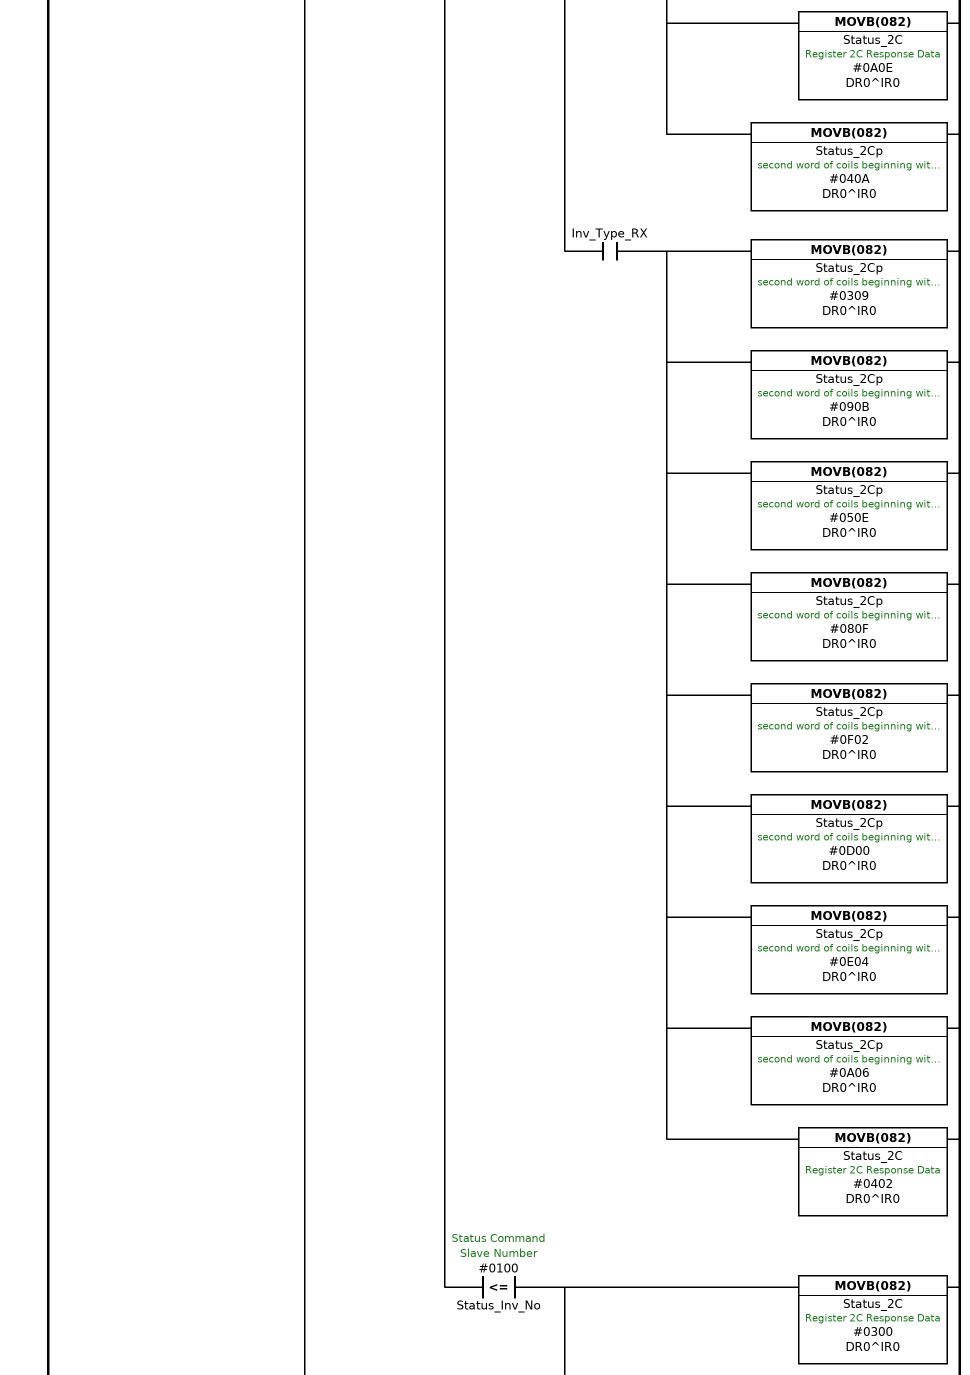
; [picture p48: FB INV002_Refresh_X31_, rungs 31-31]

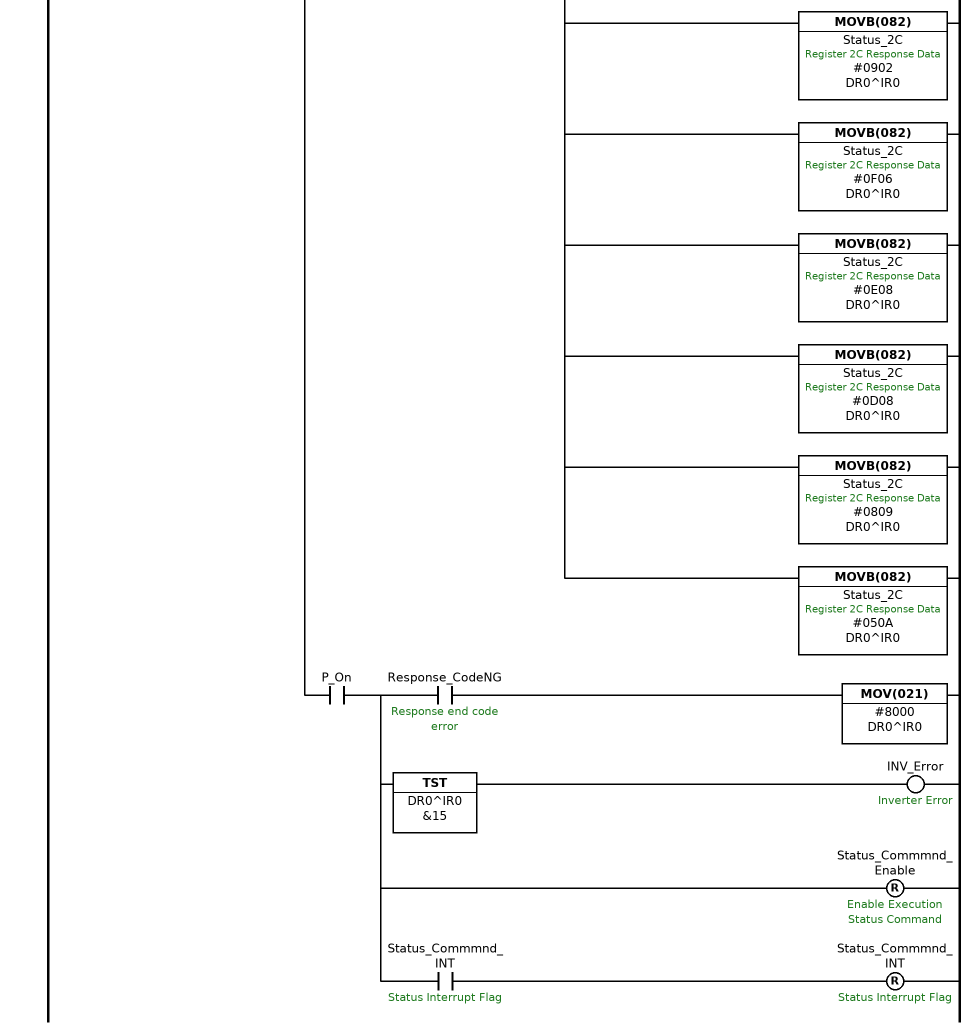
; rung 31: Generate Status Process
LD Status_Commmnd_Enable  ; Enable Execution Status Command
AND=(300) &3 Phase  ; Process Procedure
OUT TR0
AND P_On
MOV(021) Status_Inv_No Tmp_Data[0]  ; Status Command Slave Number
ANDW(034) Tmp_Data[0] #00FF Tmp_Data[0]
-(410) Tmp_Data[0] &1 Tmp_Data[0]
*(420) Tmp_Data[0] &2 Tmp_Data[0]
MOV(021) Tmp_Data[0] DR0
LD TR0
ANDNOT Response_CodeNG  ; Response end code error
OUT TR1
AND>(320) #0100 Status_Inv_No  ; Status Command Slave Number
OUT TR2
ANDNOT Inv_Type_RX
MOVB(082) Status_2C #0301 DR0^IR0  ; Register 2C Response Data
MOVB(082) Status_2C #0903 DR0^IR0  ; Register 2C Response Data
MOVB(082) Status_2C #0506 DR0^IR0  ; Register 2C Response Data
MOVB(082) Status_2C #0807 DR0^IR0  ; Register 2C Response Data
MOVB(082) Status_2C #0F0A DR0^IR0  ; Register 2C Response Data
MOVB(082) Status_2C #0D08 DR0^IR0  ; Register 2C Response Data
MOVB(082) Status_2C #0E0C DR0^IR0  ; Register 2C Response Data
MOVB(082) Status_2C #0A0E DR0^IR0  ; Register 2C Response Data
MOVB(082) Status_2Cp #040A DR0^IR0  ; second word of coils beginning with coil 1F to 2E
LD TR2
AND Inv_Type_RX
MOVB(082) Status_2Cp #0309 DR0^IR0  ; second word of coils beginning with coil 1F to 2E
MOVB(082) Status_2Cp #090B DR0^IR0  ; second word of coils beginning with coil 1F to 2E
MOVB(082) Status_2Cp #050E DR0^IR0  ; second word of coils beginning with coil 1F to 2E
MOVB(082) Status_2Cp #080F DR0^IR0  ; second word of coils beginning with coil 1F to 2E
MOVB(082) Status_2Cp #0F02 DR0^IR0  ; second word of coils beginning with coil 1F to 2E
MOVB(082) Status_2Cp #0D00 DR0^IR0  ; second word of coils beginning with coil 1F to 2E
MOVB(082) Status_2Cp #0E04 DR0^IR0  ; second word of coils beginning with coil 1F to 2E
MOVB(082) Status_2Cp #0A06 DR0^IR0  ; second word of coils beginning with coil 1F to 2E
MOVB(082) Status_2C #0402 DR0^IR0  ; Register 2C Response Data
LD TR1
AND<=(315) #0100 Status_Inv_No  ; Status Command Slave Number
MOVB(082) Status_2C #0300 DR0^IR0  ; Register 2C Response Data
MOVB(082) Status_2C #0902 DR0^IR0  ; Register 2C Response Data
MOVB(082) Status_2C #0F06 DR0^IR0  ; Register 2C Response Data
MOVB(082) Status_2C #0E08 DR0^IR0  ; Register 2C Response Data
MOVB(082) Status_2C #0D08 DR0^IR0  ; Register 2C Response Data
MOVB(082) Status_2C #0809 DR0^IR0  ; Register 2C Response Data
MOVB(082) Status_2C #050A DR0^IR0  ; Register 2C Response Data
LD TR0
AND P_On
OUT TR3
AND Response_CodeNG  ; Response end code error
MOV(021) #8000 DR0^IR0
LD TR3
ANDTST(350) DR0^IR0 &15
OUT INV_Error  ; Inverter Error
LD TR3
RSET Status_Commmnd_Enable  ; Enable Execution Status Command
AND Status_Commmnd_INT  ; Status Interrupt Flag
RSET Status_Commmnd_INT  ; Status Interrupt Flag

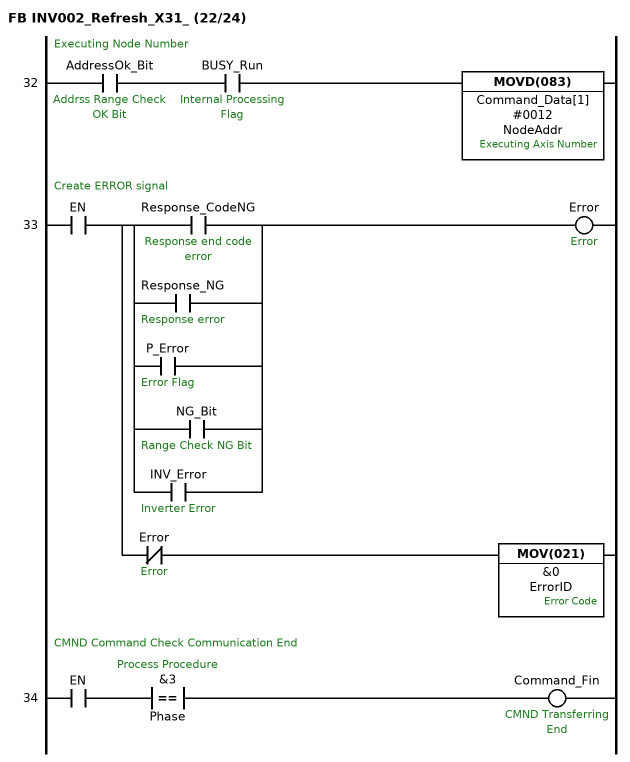
; rung 32: Executing Node Number
LD AddressOk_Bit  ; Addrss Range Check OK Bit
AND BUSY_Run  ; Internal Processing Flag
MOVD(083) Command_Data[1] #0012 NodeAddr  ; Executing Axis Number
; rung 33: Create ERROR signal
LD EN
OUT TR0
LD Response_CodeNG  ; Response end code error
OR Response_NG  ; Response error
OR P_Error  ; Error Flag
OR NG_Bit  ; Range Check NG Bit
OR INV_Error  ; Inverter Error
ANDLD
OUT Error  ; Error
LD TR0
ANDNOT Error  ; Error
MOV(021) &0 ErrorID  ; Error Code
; rung 34: CMND Command Check Communication End
LD EN
AND=(300) &3 Phase  ; Process Procedure
OUT Command_Fin  ; CMND Transferring End

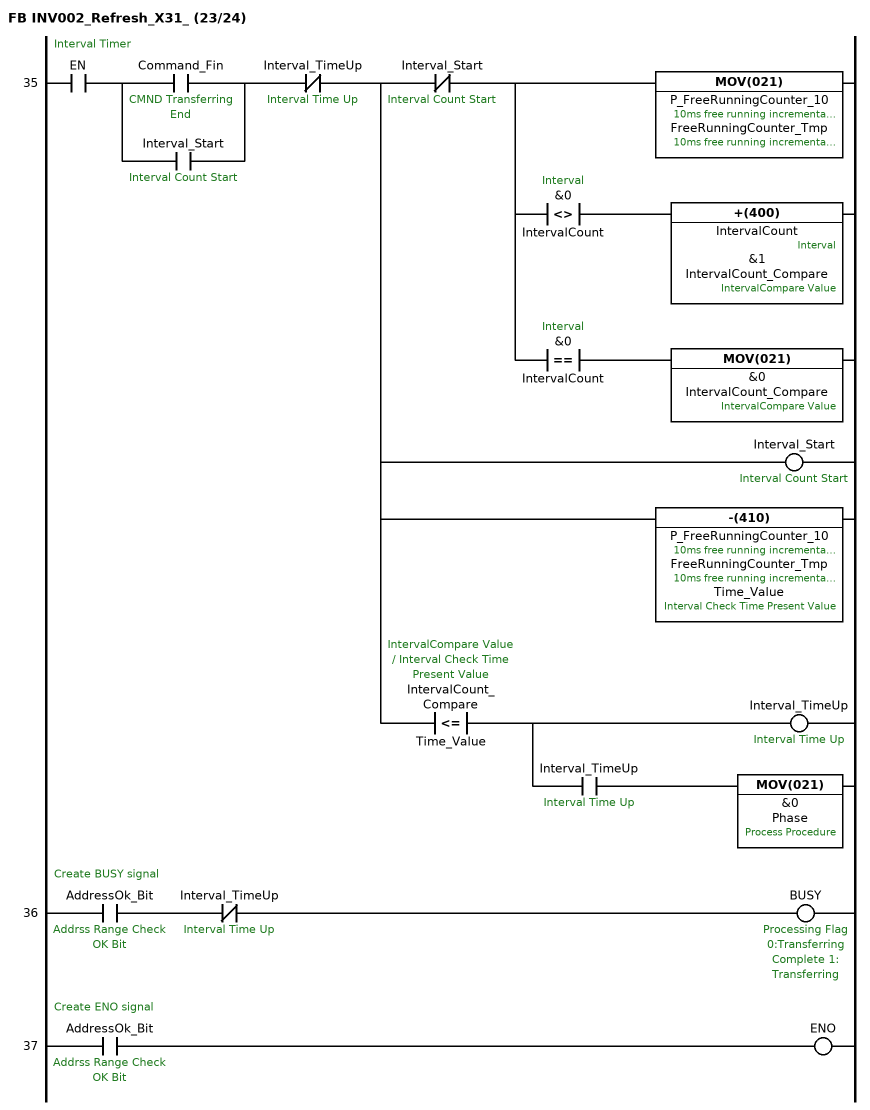
; rung 35: Interval Timer
LD EN
LD Command_Fin  ; CMND Transferring End
OR Interval_Start  ; Interval Count Start
ANDLD
ANDNOT Interval_TimeUp  ; Interval Time Up
OUT TR0
ANDNOT Interval_Start  ; Interval Count Start
OUT TR1
MOV(021) P_FreeRunningCounter_10 FreeRunningCounter_Tmp  ; 10ms free running incremental counter, 10ms free running incremental counter record
AND<>(305) &0 IntervalCount  ; Interval
+(400) IntervalCount &1 IntervalCount_Compare  ; Interval, IntervalCompare Value
LD TR1
AND=(300) &0 IntervalCount  ; Interval
MOV(021) &0 IntervalCount_Compare  ; IntervalCompare Value
LD TR0
OUT Interval_Start  ; Interval Count Start
-(410) P_FreeRunningCounter_10 FreeRunningCounter_Tmp Time_Value  ; 10ms free running incremental counter, 10ms free running incremental counter record, Interval Check Time Present Value
AND<=(315) IntervalCount_Compare Time_Value  ; IntervalCompare Value, Interval Check Time Present Value
OUT Interval_TimeUp  ; Interval Time Up
AND Interval_TimeUp  ; Interval Time Up
MOV(021) &0 Phase  ; Process Procedure
; rung 36: Create BUSY signal
LD AddressOk_Bit  ; Addrss Range Check OK Bit
ANDNOT Interval_TimeUp  ; Interval Time Up
OUT BUSY  ; Processing Flag 0:Transferring Complete 1:Transferring
; rung 37: Create ENO signal
LD AddressOk_Bit  ; Addrss Range Check OK Bit
OUT ENO

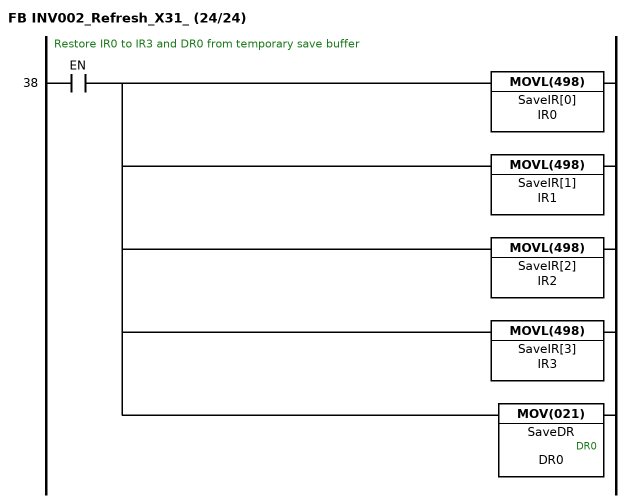
; rung 38: Restore IR0 to IR3 and DR0 from temporary save buffer
LD EN
MOVL(498) SaveIR[0] IR0
MOVL(498) SaveIR[1] IR1
MOVL(498) SaveIR[2] IR2
MOVL(498) SaveIR[3] IR3
MOV(021) SaveDR DR0  ; DR0

## Function block Новый_день
VAR_INPUT
  Day_star : UINT;
  Day_onl : UINT;
  Mon_star : UINT;
  Mon_onl : UINT;
  Day2 : UINT;
  Day3 : UINT;
  Mon2 : UINT;
  Mon3 : UINT;
END_VAR
VAR_OUTPUT
  Day_new : UINT;
  Mon_new : UINT;
  DayOut1 : UINT;
  DayOut2 : UINT;
  DayOut3 : UINT;
  MonOut1 : UINT;
  MonOut2 : UINT;
  MonOut3 : UINT;
END_VAR
	DayOut1 := Day2; DayOut2 := Day3; DayOut3 := Day_star;
	MonOut1 := Mon2; MonOut2 := Mon3; MonOut3 := Mon_star;
	Mon_new := Mon_onl;

## Function block Сброс
VAR_INPUT
  Param1 : UDINT;
  Param2 : UDINT;
  Param3 : UDINT;
  Param4 : UDINT;
  Param5 : UINT;
  Param6 : UINT;
  Param7 : UINT;
END_VAR
VAR_OUTPUT
  out1 : UDINT;
  out2 : UDINT;
  out3 : UDINT;
  out4 : UDINT;
  out5 : UINT;
  out6 : UINT;
  out7 : UINT;
END_VAR
out1 := Param1; out1 := 0;
out2 := Param2; out2 := 0;
out3 := Param3; out3 := 0;
out4 := Param4; out4 := 0;
out5 := Param5; out5 := 0;
out6 := Param6; out6 := 0;
out7 := Param7; out7 := 0;

## Function block Сброс2
VAR_INPUT
  Param1 : UINT;
  Param2 : UINT;
  Param3 : UINT;
  Param4 : UINT;
  Param5 : UINT;
  Param6 : UINT;
  Param7 : UINT;
END_VAR
VAR_OUTPUT
  out1 : UINT;
  out2 : UINT;
  out3 : UINT;
  out4 : UINT;
  out5 : UINT;
  out6 : UINT;
  out7 : UINT;
END_VAR
out1 := Param1; out1 := 0;
out2 := Param2; out2 := 0;
out3 := Param3; out3 := 0;
out4 := Param4; out4 := 0;
out5 := Param5; out5 := 0;
out6 := Param6; out6 := 0;
out7 := Param7; out7 := 0;

## Function block сдвиг_данных
VAR_INPUT
  StarStat2 : UINT;
  StarStat3 : UINT;
  Glob_stat : UDINT;
  TochOtschStat : UDINT;
END_VAR
VAR_OUTPUT
  StatOut1 : UINT;
  StatOut2 : UINT;
  StatOut3 : UINT;
  TochOtschStatNew : UDINT;
END_VAR
StatOut1 := StarStat2;
StatOut2 := StarStat3;
StatOut3 := UDINT_TO_UINT (Glob_stat - TochOtschStat);
TochOtschStatNew :=  Glob_stat;

## Function block Сдвиг_данных2
VAR_INPUT
  StarStat2 : UINT;
  StarStat3 : UINT;
  Glob_stat : UINT;
  TochOtschStat : UINT;
END_VAR
VAR_OUTPUT
  StatOut1 : UINT;
  StatOut2 : UINT;
  StatOut3 : UINT;
  TochOtschStatNew : UINT;
END_VAR
StatOut1 := StarStat2;
StatOut2 := StarStat3;
StatOut3 := Glob_stat - TochOtschStat;
TochOtschStatNew :=  Glob_stat;